FUNCTION Convert_DATE_TO_DT : BOOL
VAR_INPUT
	in : DATE;
	out : REFERENCE TO DT;
END_VAR
VAR
	converted : DT;
END_VAR

converted := DATE_TO_DT(in);

IF (DT_TO_DATE(converted) <> in) THEN
	RETURN;
END_IF

out := converted;
Convert_DATE_TO_DT := TRUE;

END_FUNCTION

(* stored: Version 1.1.0.1, ProductVersion 3.1.4024.12
   POU Convert_DATE_TO_DT: Id {1257b383-7ca1-488c-a3a4-edeed7eb95f1}, SpecialFunc None *)
